TYPE U_AXIS_NC_PARAMETER_RD :
UNION

  stState             : ARRAY[1..MAX_AXIS] OF ST_NC_PARAMETER;

  byState   AT %Q*    : ARRAY[1..MAX_AXIS] OF
                        ARRAY[1..SIZEOF(ST_NC_PARAMETER)] OF BYTE;
END_UNION
END_TYPE

(* stored: Version 1.1.0.1, ProductVersion 3.1.4026.13
   DUT U_AXIS_NC_PARAMETER_RD: Id {c5249232-3977-0772-0279-8e1635453be8} *)
